Staubli VAL3: getListItem.pgx

public program getListItem(string& x_sItem[], num x_nIndex)
  local trsf l_tTrsf
  local string l_sItem[6]
  local string l_sEvent
begin
  //
  //
  // define the item to show in the edit page Traj
  // customize an array and copy to x_sItem...
  //
  // see other traj as example
  l_sItem[0]=("Joint 1 > "+toString(".2",jEditPoint.tData[x_nIndex].jJoint.j1))
  l_sItem[1]=("Joint 2 > "+toString(".2",jEditPoint.tData[x_nIndex].jJoint.j2))
  l_sItem[2]=("Joint 3 > "+toString(".2",jEditPoint.tData[x_nIndex].jJoint.j3))
  l_sItem[3]=("Joint 4 > "+toString(".2",jEditPoint.tData[x_nIndex].jJoint.j4))
  l_sItem[4]=("Joint 5 > "+toString(".2",jEditPoint.tData[x_nIndex].jJoint.j5))
  l_sItem[5]=("Joint 6 > "+toString(".2",jEditPoint.tData[x_nIndex].jJoint.j6))
  call use:stringCopy(l_sItem,x_sItem)
end
